# EPICS StreamDevice protocol: protocols/Eco_OS-6.proto
# Eco sensors OS-6 Protocol

InTerminator = " \r \n";

Read_ozone {
    in "\_%f\_,\_%*f\_,\_%*f";
}

Read_temp {
    in "\_%*f\_,\_%f\_,\_%*f";
}

Read_humidity {
    in "\_%*f\_,\_%*f\_,\_%f";
}
